KUKA KRL program: masref_user.src, masref_user.dat

--- masref_user.src ---
&ACCESS RVP
&REL 1
&COMMENT Mastering Reference User Program
&PARAM DISKPATH = Program
DEF MasRef_USER()
END

--- masref_user.dat ---
&ACCESS RVP
&REL 1
&COMMENT Mastering Reference User Program
&PARAM DISKPATH = Program
DEFDAT  masref_user
;FOLD EXTERNAL DECLARATIONS;%{PE}%MKUKATPBASIS,%CEXT,%VCOMMON,%P
;FOLD BASISTECH EXT;%{PE}%MKUKATPBASIS,%CEXT,%VEXT,%P
EXT  BAS (BAS_COMMAND  :IN,REAL  :IN )
;ENDFOLD (BASISTECH EXT)
;FOLD USER EXT;%{E}%MKUKATPUSER,%CEXT,%VEXT,%P
;Make here your modifications

;ENDFOLD (USER EXT)
;ENDFOLD (EXTERNAL DECLERATIONS)
ENDDAT
